FUNCTION F_MaterialDensityLookup : LREAL
VAR_INPUT
    sMaterialName : T_MaxString;
END_VAR
VAR
    fbElementDensity : FB_ElementDensity;
END_VAR


fbElementDensity(
    sName := sMaterialName
);

IF fbElementDensity.bFound THEN
    F_MaterialDensityLookup := fbElementDensity.fValue;
ELSE
    F_MaterialDensityLookup := -1.0;    
END_IF

END_FUNCTION

(* stored: Version 1.1.0.1
   POU F_MaterialDensityLookup: Id {8b00a395-1007-481c-ae38-4ff8bd4b0862}, SpecialFunc None *)
